{region '#Template'}
	{attribute 'Version' := '1.2.1.0'}
	{attribute 'Tags' := '"LCID": "1031", "Text": "Universal, Sensor, BI"'}
	{attribute 'Tags' := '"LCID": "1033", "Text": "Universal, Sensor, BI"'}
	{attribute 'Using' := '"Type": "Template", "URI": "EC_AMEV"'}
	{attribute 'Using' := '"Type": "Template", "URI": "BA2_Param"'}
	{attribute 'Description' := '"LCID": "1031", "Text": "BI mit IO"'}
	{attribute 'Description' := '"LCID": "1033", "Text": "BI with IO"'}
{endregion}		 
FUNCTION_BLOCK FB_BA_SensorBinary_IO EXTENDS FB_BA_View
VAR_INPUT
END_VAR
VAR_INPUT CONSTANT
	Input					: FB_BA_BI_IO;		
END_VAR
VAR_OUTPUT
	bPresentValue			: BOOL;	
END_VAR
VAR
END_VAR

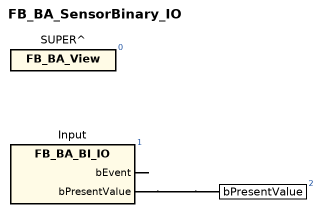
SUPER^(); // FB_BA_View
Input(); // FB_BA_BI_IO
bPresentValue := Input.bPresentValue;

METHOD FB_init : BOOL
VAR_INPUT
	bInitRetains : BOOL; // if TRUE, the retain variables are initialized (warm start / cold start)
	bInCopyCode : BOOL;  // if TRUE, the instance afterwards gets moved into the copy code (online change)
END_VAR
Input.iParent						:= THIS^;
Input.iLabel						:= LblUniFieldDevice.SensorBinary_Input;	
Input.sObjectName					:= '{Idx=01}';	
Input.sDeviceType					:= '';
Input.bEnOutOfService				:= FALSE;
Input.ePolarity						:= E_BA_Polarity.eReverse;
Input.sActiveText 					:= txtEvent_Triggered;
Input.sInactiveText 				:= txtEvent_Normal;
Input.nStateChangeCount				:= 0;
Input.nActiveTimeElapsed			:= 0;
Input.nEventClassID					:= EC_ID.NC30;
Input.stTimeDelay.nToNormal			:= BA2_Param.nDefTimeDelay_ToNormal;
Input.stTimeDelay.nToAbnormal		:= BA2_Param.nDefTimeDelay_ToAbnormal;
Input.bAlarmValue					:= TRUE;
Input.bAcknowledgeRm				:= FALSE;		
Input.aEventTransitionText[1]		:= txtEvent_Triggered;
Input.aEventTransitionText[2]		:= txtEvent_Error;
Input.aEventTransitionText[3]		:= txtEvent_Normal;
Input.bEventDetectionEnable			:= TRUE;
Input.aEventEnable[1]				:= TRUE;			//	to_offnormal
Input.aEventEnable[2]				:= TRUE;			//	to_fault
Input.aEventEnable[3]				:= TRUE;			//	to_normal
Input.eEnPlantLock					:= E_BA_LockPriority.eNoLock;
END_METHOD

END_FUNCTION_BLOCK

(* stored: Version 1.1.0.1, ProductVersion 3.1.4024.9
   POU FB_BA_SensorBinary_IO: Id {351c177c-9a4e-4a8e-aadf-6eb9f0c15671}, SpecialFunc None
   Method FB_init: Id {5723bee6-d90c-439c-b89b-12c34b11abea} *)
